Staubli VAL3: onEdit.pgx

public program onEdit(string& x_sItem[])
  local string l_sPath
  local num i
  local string l_sItem
  local num l_nSize
  local TrajectoryItem l_tTraj
  local num l_nResult
  local string l_sPoint
begin
  // DEFINE YOUR ITEM
  call getTrajType(saveData:sTrajTypeUsing)
  // load the trajectory
  call load(x_sItem,l_nResult)
  if find(x_sItem,"@")==-1
    // load the page viewTraj
    l_sPath="Disk://trajectory/page_viewTraj"
    // give back the path
    x_sItem[1]=x_sItem
    x_sItem=l_sPath
  endIf
end
